{attribute 'qualified_only'}
{attribute 'strict'}
TYPE E_STM_QLearning :
(
	init := 0,
	reset,
	resetWaitOK,
	step,
	stepOK,
	compute,
	computeOK,
	playEnvironment,
	donePlayingEnvironment
);
END_TYPE

(* stored: Version 1.1.0.1, ProductVersion 3.1.4024.12
   DUT E_STM_QLearning: Id {78f8b589-5c3d-404d-b48a-29788f28b0d9} *)
